FUNCTION_BLOCK KIN_CALCTRAFO_AXPOS_PARAM
VAR_INPUT
	In														: 	ARRAY[1..8] OF LREAL;
	Out														: 	ARRAY[1..8] OF LREAL;
	MetaInfoIn												:	U_KinMetaInfo;
	MetaInfoOut												:	U_KinMetaInfo;
END_VAR
VAR_OUTPUT
END_VAR
VAR
END_VAR

METHOD delete : BOOL
VAR_INPUT
END_VAR
MEMSET(ADR(In),0,SIZEOF(In));
MEMSET(ADR(Out),0,SIZEOF(Out));
delete	:= TRUE;
END_METHOD

END_FUNCTION_BLOCK

(* stored: Version 1.1.0.1, ProductVersion 3.1.4024.6
   POU KIN_CALCTRAFO_AXPOS_PARAM: Id {8b73be1b-7e19-4cca-ba2f-e340d072801f}, SpecialFunc None
   Method delete: Id {56d95162-190c-4093-b0d7-4b2962333dc7} *)
